FUNCTION_BLOCK fbIO_DigitalOutput
VAR_INPUT
	iInMode:INT;		(*global mode input*)
	bInEstop:BOOL;		(* Emergency stop input 0=Estop Active*)
	bInEnable:BOOL;		(*Interlock for the digital output. If this bit is false, then output will be 0*)
	bInCommand:BOOL;	(*The command to the digital output*)
END_VAR
VAR_OUTPUT
	bOutAuto:BOOL;		(*Block in auto mode*)
	bOutCommand:BOOL;	(*Command to digital output*)
END_VAR
VAR_IN_OUT
	HMI_IO_DigitalOutput:stHMI_DigitalOutput;
END_VAR
VAR
	bTempOutCommand:BOOL;
	bSetHMICommandsOFF:BOOL;
END_VAR

(*control bOut based on the global input and HMI input mode*)
(*if in independant mode allow control of the output based on HMI commands (MANUAL) AND digital input (AUTO)*)
IF iInMode=10 THEN
	//if HMI requests manual mode 
	IF HMI_IO_DigitalOutput.iMode=2 THEN
		bOutAuto:=0;
		bSetHMICommandsOFF:=0;
		IF HMI_IO_DigitalOutput.bPBEN_On AND HMI_IO_DigitalOutput.bPB_On THEN
			bTempOutCommand:=1;
		ELSIF HMI_IO_DigitalOutput.bPBEN_Off AND HMI_IO_DigitalOutput.bPB_Off THEN
			bTempOutCommand:=0;
		END_IF
	ELSE
		bTempOutCommand:=bInCommand;   /// auto output
		bOutAuto:=1;
		bSetHMICommandsOFF:=1;
	END_IF
ELSE
	bTempOutCommand:=bInCommand;   /// auto output
	bSetHMICommandsOFF:=1;
	bOutAuto:=1;
END_IF

bOutCommand := bTempOutCommand AND  bInEnable AND bInEstop;//allow output when interlocked and Estop ok

HMI_IO_DigitalOutput.bCommandAuto:=bInCommand;
HMI_IO_DigitalOutput.bCommand:=bTempOutCommand;
HMI_IO_DigitalOutput.bInterlock:=bInEnable;

IF bSetHMICommandsOFF THEN
	HMI_IO_DigitalOutput.iMode:=1;
	HMI_IO_DigitalOutput.bPBEN_On:=0;
	HMI_IO_DigitalOutput.bPBEN_Off:=0;
	HMI_IO_DigitalOutput.bPB_On:=0;
	HMI_IO_DigitalOutput.bPB_Off:=0;
END_IF

END_FUNCTION_BLOCK

(* stored: Version 1.1.0.1, ProductVersion 3.1.4024.11
   POU fbIO_DigitalOutput: Id {3a95440e-cc1a-4e61-a388-df1954919aa5}, SpecialFunc None *)
